FUNCTION CreateJsonDocumentManual : STRING(1000)
VAR_INPUT
	MaterialID : STRING;
	CheckFor : STRING;
	CameraNumber : INT;
END_VAR
VAR
	fbJson : FB_JsonSaxWriter;
END_VAR

fbJson.StartObject();

fbJson.AddKey('MaterialID');
fbJson.AddString(MaterialID);

fbJson.AddKey('CheckFor');
fbJson.AddString(CheckFor);

fbJson.AddKey('CameraNumber');
fbJson.AddString(CameraNumber);

//below are keys for VisionPC to write to
fbJson.AddKey('SuccessFlag');
fbJson.AddKey('OrientAdjustX');
fbJson.AddKey('OrientAdjustY');
fbJson.AddKey('OrientAdjustX');

fbJson.EndObject();

CreateJsonDocumentManual := fbJson.GetDocument();

END_FUNCTION

(* stored: Version 1.1.0.1, ProductVersion 3.1.4024.11
   POU CreateJsonDocumentManual: Id {e92a94bb-6357-4e2e-aceb-ff7bdd64c4c4}, SpecialFunc None *)
